INTERFACE IPAControlModule EXTENDS IACComponent

PROPERTY AllocatedByFunction : IPAProcessFunction
GET
END_GET
SET
END_SET
END_PROPERTY

PROPERTY AllocatedByWay : BOOL
GET
END_GET
END_PROPERTY

METHOD HasPointReachedOffPosition : BOOL
VAR_INPUT
	point : IACPoint;
END_VAR
END_METHOD

METHOD HasPointReachedOnPosition : BOOL
VAR_INPUT
	point : IACPoint;
END_VAR
END_METHOD

PROPERTY RoutingStateFromSource : PARoutingState
GET
END_GET
END_PROPERTY

PROPERTY RoutingStateOfPredecessors : PARoutingState
GET
END_GET
END_PROPERTY

PROPERTY RoutingStateOfSuccessors : PARoutingState
GET
END_GET
END_PROPERTY

PROPERTY RoutingStateThis : PARoutingState
GET
END_GET
END_PROPERTY

PROPERTY RoutingStateToTarget : PARoutingState
GET
END_GET
END_PROPERTY

END_INTERFACE

(* stored: Version 1.1.0.1, ProductVersion 3.1.4020.12
   Itf IPAControlModule: Id {11d215b8-d751-4464-8b4c-6653f7fff126}
   Property AllocatedByFunction: Id {c981204d-1045-467b-b7c9-989c89bf80f0}
   Get Get: Id {837f1910-dad3-4dcc-9e8a-69fa7f2c6b60}
   Set Set: Id {206e6151-63f2-4a3a-8ce5-eccc42a2a3b8}
   Property AllocatedByWay: Id {19ce5e44-867a-42d7-804c-5b3225c131e8}
   Get Get: Id {ed95a34b-8b3c-4b86-8947-f67065824331}
   Method HasPointReachedOffPosition: Id {f6dcab94-a511-404f-aa01-373fa4d1c568}
   Method HasPointReachedOnPosition: Id {5407737d-b567-4913-b43a-2daff21d7296}
   Property RoutingStateFromSource: Id {9e4a0f87-1261-4da0-b200-114ae5a91ae1}
   Get Get: Id {f88aeba7-d031-406a-8218-583506b452e2}
   Property RoutingStateOfPredecessors: Id {13929c78-e921-4a3b-a903-4c9759f49c81}
   Get Get: Id {ad4c2a16-ba2d-4888-8b69-6d820e7ff233}
   Property RoutingStateOfSuccessors: Id {e82ed9f4-4053-431c-ac03-722a1685adb1}
   Get Get: Id {9f90f9ac-f844-42d6-b400-919bfd5057cd}
   Property RoutingStateThis: Id {c4804d5b-bfba-45c1-94fd-051ae44bf6b2}
   Get Get: Id {a95127b3-74f6-409e-b6fd-aca3c77b57e6}
   Property RoutingStateToTarget: Id {2a13bca0-010a-413e-be4e-518ee37ae078}
   Get Get: Id {f104dd49-dc46-4a9b-9391-04424d079467} *)
